(* PLC project bilfabriken.project, CODESYS CODESYS V3.5 SP4 Patch 3 *)
(* stored: creationDateTime 2015-02-05T18:21:50.255309, modificationDateTime 2015-02-05T17:25:27.6708362 *)

(* Exempel: Generera slumptal mellan 1 ooch 10. randNext : ULINT := 42; x : uint := rand(1,10) Ger ett slumptal mellan lower och upper Kräver att man har definierat en variabel randNext:ULINT:=<ett frö>; Ref: Bilting, U. Vägen Till C. Studentlitteratur. 2011. *)
FUNCTION rand : UINT
  VAR_INPUT
    lower : UINT;
    upper : UINT;
  END_VAR
  VAR
    range : UINT := ((upper - lower) + 1);
    interval : UINT := (c4 / range);
    preRand : UINT;
  END_VAR
  VAR CONSTANT
    c1 : UDINT := 1103515245;
    c2 : UINT := 12345;
    c3 : UDINT := 65536;
    c4 : UINT := 32768;
  END_VAR

            randNext := randNext * c1 + c2;
preRand := ULINT_TO_UINT((randNext/c3) MOD c4);
IF interval > 0 THEN
	rand := (preRand+lower*interval-1)/interval; 
ELSE
	rand := preRand;
END_IF;
RETURN;
          
END_FUNCTION

PROGRAM TestRand
  VAR
    randNext : ULINT := 42;
    x : UINT;
  END_VAR

            x := rand(1,10);
          
END_PROGRAM
